FUNCTION_BLOCK SPLIT_AL_INTO_AQ (* this Function splits the 32 AQ (QUARTER) adapters from a AL (LWORD) *)
  (* Standard: 61499-2; Description: Copyright (c) 2026 Meisterschulen am Ostbahnhof SPDX-License-Identifier: EPL-2.0 *)
  (* Version 1.0, 2026-05-16, Franz Höpfinger, Meisterschulen am Ostbahnhof, initial API and implementation and/or initial documentation *)
  PACKAGE adapter::splitting;
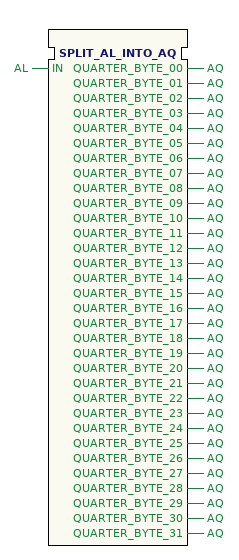
  SOCKETS
    IN : adapter::types::unidirectional::AL; (* LWORD Input *)
  END_SOCKETS
  PLUGS
    QUARTER_BYTE_00 : adapter::types::unidirectional::AQ; (* Quarter 0 *)
    QUARTER_BYTE_01 : adapter::types::unidirectional::AQ; (* Quarter 1 *)
    QUARTER_BYTE_02 : adapter::types::unidirectional::AQ; (* Quarter 2 *)
    QUARTER_BYTE_03 : adapter::types::unidirectional::AQ; (* Quarter 3 *)
    QUARTER_BYTE_04 : adapter::types::unidirectional::AQ; (* Quarter 4 *)
    QUARTER_BYTE_05 : adapter::types::unidirectional::AQ; (* Quarter 5 *)
    QUARTER_BYTE_06 : adapter::types::unidirectional::AQ; (* Quarter 6 *)
    QUARTER_BYTE_07 : adapter::types::unidirectional::AQ; (* Quarter 7 *)
    QUARTER_BYTE_08 : adapter::types::unidirectional::AQ; (* Quarter 8 *)
    QUARTER_BYTE_09 : adapter::types::unidirectional::AQ; (* Quarter 9 *)
    QUARTER_BYTE_10 : adapter::types::unidirectional::AQ; (* Quarter 10 *)
    QUARTER_BYTE_11 : adapter::types::unidirectional::AQ; (* Quarter 11 *)
    QUARTER_BYTE_12 : adapter::types::unidirectional::AQ; (* Quarter 12 *)
    QUARTER_BYTE_13 : adapter::types::unidirectional::AQ; (* Quarter 13 *)
    QUARTER_BYTE_14 : adapter::types::unidirectional::AQ; (* Quarter 14 *)
    QUARTER_BYTE_15 : adapter::types::unidirectional::AQ; (* Quarter 15 *)
    QUARTER_BYTE_16 : adapter::types::unidirectional::AQ; (* Quarter 16 *)
    QUARTER_BYTE_17 : adapter::types::unidirectional::AQ; (* Quarter 17 *)
    QUARTER_BYTE_18 : adapter::types::unidirectional::AQ; (* Quarter 18 *)
    QUARTER_BYTE_19 : adapter::types::unidirectional::AQ; (* Quarter 19 *)
    QUARTER_BYTE_20 : adapter::types::unidirectional::AQ; (* Quarter 20 *)
    QUARTER_BYTE_21 : adapter::types::unidirectional::AQ; (* Quarter 21 *)
    QUARTER_BYTE_22 : adapter::types::unidirectional::AQ; (* Quarter 22 *)
    QUARTER_BYTE_23 : adapter::types::unidirectional::AQ; (* Quarter 23 *)
    QUARTER_BYTE_24 : adapter::types::unidirectional::AQ; (* Quarter 24 *)
    QUARTER_BYTE_25 : adapter::types::unidirectional::AQ; (* Quarter 25 *)
    QUARTER_BYTE_26 : adapter::types::unidirectional::AQ; (* Quarter 26 *)
    QUARTER_BYTE_27 : adapter::types::unidirectional::AQ; (* Quarter 27 *)
    QUARTER_BYTE_28 : adapter::types::unidirectional::AQ; (* Quarter 28 *)
    QUARTER_BYTE_29 : adapter::types::unidirectional::AQ; (* Quarter 29 *)
    QUARTER_BYTE_30 : adapter::types::unidirectional::AQ; (* Quarter 30 *)
    QUARTER_BYTE_31 : adapter::types::unidirectional::AQ; (* Quarter 31 *)
  END_PLUGS
END_FUNCTION_BLOCK
